PROGRAM MAIN
VAR
	fbUPS : FB_S_UPS_CX51x0;
	SPDM_2PASS: E_PersistentMode;
END_VAR

actUps();

ACTION actUps:
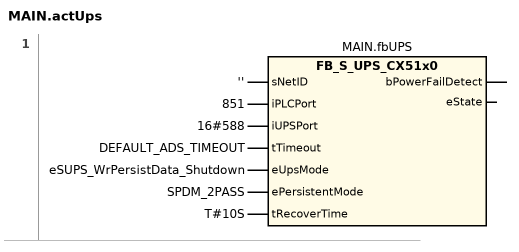
// NETWORK 1
MAIN.fbUPS(
    sNetID := '',
    iPLCPort := 851,
    iUPSPort := 16#588,
    tTimeout := DEFAULT_ADS_TIMEOUT,
    eUpsMode := eSUPS_WrPersistData_Shutdown,
    ePersistentMode := SPDM_2PASS,
    tRecoverTime := T#10S); // FB_S_UPS_CX51x0
END_ACTION

END_PROGRAM

(* stored: Version 1.1.0.1, ProductVersion 3.1.4024.12
   POU MAIN: Id {b2d3b134-95c6-4907-b8f4-f414088f0508}, SpecialFunc None
   Action actUps: Id {0f4e6d04-e0ff-4659-8385-d0d67aad2843} *)
